(* IEC 61131-3 sources: JaccoSigma/tempclass/Class/SramCheck, 1 file *)

(* ---- SramCheck.st ---- *)
(*!
<Class
	Name               = "SramCheck"
	Revision           = "0.0"
	RealtimeTask       = "false"
	CyclicTask         = "false"
	BackgroundTask     = "true"
	Sigmatek           = "false"
	OSInterface        = "false"
	HighPriority       = "false"
	Automatic          = "false"
	UpdateMode         = "Prescan"
	SharedCommandTable = "true"
	Objectsize         = "(392,120)">
	<Channels>
		<Server Name="ClassSvr" Visualized="true" Remotely="true" Initialize="false" WriteProtected="false" Retentive="SRam"/>
		<Server Name="Data" Class="StringRAM" Visualized="true" Remotely="true" Initialize="true" WriteProtected="false" Retentive="false"/>
		<Server Name="Data0" Class="StringRAM" Visualized="true" Remotely="true" Initialize="true" WriteProtected="false" Retentive="false"/>
		<Server Name="Data1" Class="StringRAM" Visualized="true" Remotely="true" Initialize="true" WriteProtected="false" Retentive="false"/>
		<Server Name="Data2" Class="StringRAM" Visualized="true" Remotely="true" Initialize="true" WriteProtected="false" Retentive="false"/>
		<Server Name="Data3" Class="Ram" Visualized="true" Remotely="true" Initialize="true" WriteProtected="false" Retentive="false"/>
		<Server Name="Data4" Class="Ram" Visualized="true" Remotely="true" Initialize="true" WriteProtected="false" Retentive="false"/>
		<Server Name="m_udLength" Class="RAMex" Visualized="true" Remotely="true" Initialize="true" WriteProtected="false" Retentive="false" Comment="length of the data buffer"/>
		<Server Name="RAMexDo" Visualized="true" Remotely="true" Initialize="false" WriteProtected="false" Retentive="false"/>
		<Server Name="Server" Visualized="true" Remotely="true" Initialize="false" WriteProtected="false" Retentive="SRam"/>
		<Server Name="Server0" Visualized="true" Remotely="true" Initialize="false" WriteProtected="false" Retentive="SRam"/>
		<Server Name="Server1" Visualized="true" Remotely="true" Initialize="false" WriteProtected="false" Retentive="File"/>
		<Server Name="Server2" Visualized="true" Remotely="true" Initialize="false" WriteProtected="false" Retentive="File"/>
		<Server Name="Server3" Visualized="true" Remotely="true" Initialize="false" WriteProtected="false" Retentive="File"/>
		<Client Name="Ram1" Required="true" Internal="true"/>
		<Client Name="Ram2" Required="true" Internal="true"/>
		<Client Name="RAMex1" Required="true" Internal="true"/>
	</Channels>
	<Network Name="SramCheck">
		<!-- List of Components in this network -->
		<Components>
			<Object
				Name       = "Ram1"
				Class      = "Ram"
				Position   = "(60,1410)"
				Visualized = "true"
				Remotely   = "true">
				<Channels>
					<Server Name="Data"/>
				</Channels>
			</Object>
			<Object
				Name       = "Ram2"
				Class      = "Ram"
				Position   = "(60,1560)"
				Visualized = "true"
				Remotely   = "true">
				<Channels>
					<Server Name="Data"/>
				</Channels>
			</Object>
			<Object
				Name       = "RAMex1"
				Class      = "RAMex"
				Position   = "(60,1740)"
				Visualized = "true"
				Remotely   = "true">
				<Channels>
					<Server Name="m_udLength"/>
					<Client Name="MultiTask"/>
					<Client Name="ThreadSafe" Value="0"/>
					<Client Name="UseFile"/>
				</Channels>
			</Object>
		</Components>
		<Comments>
		</Comments>
		<!-- List of Connections in this network -->
		<Connections>
			<Connection Source="this.Ram1" Destination="Ram1.Data"/>
			<Connection Source="this.Ram2" Destination="Ram2.Data"/>
			<Connection Source="this.Data3" Destination="Ram1.Data" Vertices="(532,810),(600,1500),(360,1500),"/>
			<Connection Source="this.Data4" Destination="Ram2.Data" Vertices="(532,870),(600,1650),(360,1650),"/>
			<Connection Source="this.RAMex1" Destination="RAMex1.m_udLength"/>
			<Connection Source="this.m_udLength" Destination="RAMex1.m_udLength" Vertices="(532,930),(360,1830),"/>
		</Connections>
		<!-- Headerfiles -->
		<Options>
		</Options>
	</Network>
</Class>
*)
SramCheck : CLASS
  //Servers:
	ClassSvr 	: SvrChCmd_DINT;
	Server 	: SvrCh_DINT;
	Server0 	: SvrCh_DINT;
	Server1 	: SvrCh_DINT;
	Server2 	: SvrCh_DINT;
	Server3 	: SvrCh_DINT;
	Data 	: SvrChCmd_UDINT;
	Data0 	: SvrChCmd_UDINT;
	Data1 	: SvrChCmd_UDINT;
	Data2 	: SvrChCmd_UDINT;
	Data3 	: SvrChCmd_DINT;
	Data4 	: SvrChCmd_DINT;
	m_udLength 	: SvrChCmd_UDINT;
	RAMexDo 	: SvrCh_DINT;
  //Clients:
	Ram1 	: CltChCmd_Ram;
	Ram2 	: CltChCmd_Ram;
	RAMex1 	: CltChCmd_RAMex;
  //Variables:
  //Functions:

	FUNCTION VIRTUAL GLOBAL Init;

	FUNCTION VIRTUAL GLOBAL Background
		VAR_INPUT
			EAX 	: UDINT;
		END_VAR
		VAR_OUTPUT
			state (EAX) 	: UDINT;
		END_VAR;

	FUNCTION VIRTUAL GLOBAL Data::Read
		VAR_OUTPUT
			output (EAX) 	: UDINT;
		END_VAR;

	FUNCTION VIRTUAL GLOBAL Data::Write
		VAR_INPUT
			input (EAX) 	: UDINT;
		END_VAR
		VAR_OUTPUT
			result (EAX) 	: UDINT;
		END_VAR;

	FUNCTION VIRTUAL GLOBAL Data0::Read
		VAR_OUTPUT
			output (EAX) 	: UDINT;
		END_VAR;

	FUNCTION VIRTUAL GLOBAL Data0::Write
		VAR_INPUT
			input (EAX) 	: UDINT;
		END_VAR
		VAR_OUTPUT
			result (EAX) 	: UDINT;
		END_VAR;

	FUNCTION VIRTUAL GLOBAL Data1::Read
		VAR_OUTPUT
			output (EAX) 	: UDINT;
		END_VAR;

	FUNCTION VIRTUAL GLOBAL Data1::Write
		VAR_INPUT
			input (EAX) 	: UDINT;
		END_VAR
		VAR_OUTPUT
			result (EAX) 	: UDINT;
		END_VAR;

	FUNCTION VIRTUAL GLOBAL Data2::Read
		VAR_OUTPUT
			output (EAX) 	: UDINT;
		END_VAR;

	FUNCTION VIRTUAL GLOBAL Data2::Write
		VAR_INPUT
			input (EAX) 	: UDINT;
		END_VAR
		VAR_OUTPUT
			result (EAX) 	: UDINT;
		END_VAR;

	FUNCTION VIRTUAL GLOBAL Data3::Read
		VAR_OUTPUT
			output (EAX) 	: DINT;
		END_VAR;

	FUNCTION VIRTUAL GLOBAL Data3::Write
		VAR_INPUT
			input (EAX) 	: DINT;
		END_VAR
		VAR_OUTPUT
			result (EAX) 	: DINT;
		END_VAR;

	FUNCTION VIRTUAL GLOBAL Data4::Read
		VAR_OUTPUT
			output (EAX) 	: DINT;
		END_VAR;

	FUNCTION VIRTUAL GLOBAL Data4::Write
		VAR_INPUT
			input (EAX) 	: DINT;
		END_VAR
		VAR_OUTPUT
			result (EAX) 	: DINT;
		END_VAR;

	FUNCTION VIRTUAL GLOBAL m_udLength::Read
		VAR_OUTPUT
			output (EAX) 	: UDINT;
		END_VAR;

	FUNCTION VIRTUAL GLOBAL m_udLength::Write
		VAR_INPUT
			input (EAX) 	: UDINT;
		END_VAR
		VAR_OUTPUT
			result (EAX) 	: UDINT;
		END_VAR;

	FUNCTION VIRTUAL GLOBAL RAMexDo::Write
		VAR_INPUT
			input (EAX) 	: DINT;
		END_VAR
		VAR_OUTPUT
			result (EAX) 	: DINT;
		END_VAR;
  //Tables:
	FUNCTION @STD
		VAR_OUTPUT
			ret_code	: CONFSTATES;
		END_VAR;
	FUNCTION GLOBAL TAB @CT_;
END_CLASS;

#pragma using Ram
#pragma using RAMex

FUNCTION VIRTUAL GLOBAL SramCheck::Data::Read
	VAR_OUTPUT
		output (EAX) 	: UDINT;
	END_VAR

	Data := StringRAM1.Data.Read();
	output := Data;

END_FUNCTION

FUNCTION VIRTUAL GLOBAL SramCheck::Data::Write
	VAR_INPUT
		input (EAX) 	: UDINT;
	END_VAR
	VAR_OUTPUT
		result (EAX) 	: UDINT;
	END_VAR

	Data := input;
	result := (StringRAM1.Data.Write(Data))$UDINT;

END_FUNCTION

FUNCTION VIRTUAL GLOBAL SramCheck::Data0::Read
	VAR_OUTPUT
		output (EAX) 	: UDINT;
	END_VAR

	Data0 := StringRAM2.Data.Read();
	output := Data0;

END_FUNCTION

FUNCTION VIRTUAL GLOBAL SramCheck::Data0::Write
	VAR_INPUT
		input (EAX) 	: UDINT;
	END_VAR
	VAR_OUTPUT
		result (EAX) 	: UDINT;
	END_VAR

	Data0 := input;
	result := (StringRAM2.Data.Write(Data0))$UDINT;

END_FUNCTION

FUNCTION VIRTUAL GLOBAL SramCheck::Data1::Read
	VAR_OUTPUT
		output (EAX) 	: UDINT;
	END_VAR

	Data1 := StringRAM3.Data.Read();
	output := Data1;

END_FUNCTION

FUNCTION VIRTUAL GLOBAL SramCheck::Data1::Write
	VAR_INPUT
		input (EAX) 	: UDINT;
	END_VAR
	VAR_OUTPUT
		result (EAX) 	: UDINT;
	END_VAR

	Data1 := input;
	result := (StringRAM3.Data.Write(Data1))$UDINT;

END_FUNCTION

FUNCTION VIRTUAL GLOBAL SramCheck::Data2::Read
	VAR_OUTPUT
		output (EAX) 	: UDINT;
	END_VAR

	Data2 := StringRAM4.Data.Read();
	output := Data2;

END_FUNCTION

FUNCTION VIRTUAL GLOBAL SramCheck::Data2::Write
	VAR_INPUT
		input (EAX) 	: UDINT;
	END_VAR
	VAR_OUTPUT
		result (EAX) 	: UDINT;
	END_VAR

	Data2 := input;
	result := (StringRAM4.Data.Write(Data2))$UDINT;

END_FUNCTION

FUNCTION VIRTUAL GLOBAL SramCheck::Data3::Read
	VAR_OUTPUT
		output (EAX) 	: DINT;
	END_VAR

	Data3 := Ram1.Data.Read();
	output := Data3;

END_FUNCTION

FUNCTION VIRTUAL GLOBAL SramCheck::Data3::Write
	VAR_INPUT
		input (EAX) 	: DINT;
	END_VAR
	VAR_OUTPUT
		result (EAX) 	: DINT;
	END_VAR

	Data3 := input;
	result := (Ram1.Data.Write(Data3))$DINT;

END_FUNCTION

FUNCTION VIRTUAL GLOBAL SramCheck::Data4::Read
	VAR_OUTPUT
		output (EAX) 	: DINT;
	END_VAR

	Data4 := Ram2.Data.Read();
	output := Data4;

END_FUNCTION

FUNCTION VIRTUAL GLOBAL SramCheck::Data4::Write
	VAR_INPUT
		input (EAX) 	: DINT;
	END_VAR
	VAR_OUTPUT
		result (EAX) 	: DINT;
	END_VAR

	Data4 := input;
	result := (Ram2.Data.Write(Data4))$DINT;

END_FUNCTION

FUNCTION VIRTUAL GLOBAL SramCheck::m_udLength::Read
	VAR_OUTPUT
		output (EAX) 	: UDINT;
	END_VAR

	m_udLength := RAMex1.m_udLength.Read();
	output := m_udLength;

END_FUNCTION

FUNCTION VIRTUAL GLOBAL SramCheck::m_udLength::Write
	VAR_INPUT
		input (EAX) 	: UDINT;
	END_VAR
	VAR_OUTPUT
		result (EAX) 	: UDINT;
	END_VAR

	m_udLength := input;
	result := (RAMex1.m_udLength.Write(m_udLength))$UDINT;

END_FUNCTION

FUNCTION VIRTUAL GLOBAL SramCheck::Init

  if _FirstScan = TRUE then

    if RAMex1.m_udLength = 0 then
      RAMex1.SetSize(udSize:=sizeof(RAMexDo));
    else
      RAMex1.GetData(pData:=#RAMexDo$USINT);
    end_if;

  end_if;

END_FUNCTION

FUNCTION VIRTUAL GLOBAL SramCheck::Background
	VAR_INPUT
		EAX 	: UDINT;
	END_VAR
	VAR_OUTPUT
		state (EAX) 	: UDINT;
	END_VAR

	state := READY;

END_FUNCTION

FUNCTION VIRTUAL GLOBAL SramCheck::RAMexDo::Write
	VAR_INPUT
		input (EAX) 	: DINT;
	END_VAR
	VAR_OUTPUT
		result (EAX) 	: DINT;
	END_VAR

	RAMexDo := input;

  if input = 0 then
    RAMex1.GetData(pData:=#RAMexDo$USINT);
  else
    RAMex1.SetData(pData:=#RAMexDo$USINT);
  end_if;

	result := RAMexDo;

END_FUNCTION
